FUNCTION FC_AnalogRead : REAL
VAR_INPUT
	SelectData : WORD;
	SelectRange : INT;
END_VAR
VAR
	Transdata : REAL;
END_VAR

Transdata := WORD_TO_REAL(selectData);
// FC_AnalogRead :=(Transdata*SelectRange)/32767;
FC_AnalogRead :=(Transdata/32767)*SelectRange;

END_FUNCTION

(* stored: Version 1.1.0.1, ProductVersion 3.1.4024.13
   POU FC_AnalogRead: Id {ee5eb385-9e3f-4368-8507-3c0800cdfdf1}, SpecialFunc None *)
